FUNCTION GET_MIN_DISTANCE_NODE : INT
VAR_INPUT
	aDistances : ARRAY[1..24] OF INT;
	aVisited : ARRAY[1..24] OF BOOL;
END_VAR
VAR
	i, nMinIndex, nMinDistance : INT;
END_VAR

nMinIndex := -1;
nMinDistance := GLOBALS.nAVeryLargeNumber;

FOR i := 1 TO 24 DO
	IF NOT (aVisited[i]) AND (aDistances[i] <= nMinDistance) THEN
		nMinDistance := aDistances[i];
		nMinIndex := i;
	END_IF
END_FOR

GET_MIN_DISTANCE_NODE := nMinIndex;

END_FUNCTION

(* stored: Version 1.1.0.1, ProductVersion 3.1.4024.12
   POU GET_MIN_DISTANCE_NODE: Id {8e711ae3-9854-4a55-b940-55e63fc297b4}, SpecialFunc None *)
